PROGRAM main
VAR
	MODBEE_HW_INPUTS0 : MODBEE_HW_INPUTS;
	MODBEE_HW_OUTPUTS0 : MODBEE_HW_OUTPUTS;
	start : bool;
	stop : bool;
	run : bool;
	MODBUS_WRITE0 : MODBUS_WRITE;
	MB_SLAVE_DO01 : bool;
	MB_SLAVE_DO02 : bool;
	MB_SLAVE_DO03 : bool;
	MB_SLAVE_DO04 : bool;
	MB_SLAVE_DO05 : bool;
	MB_SLAVE_DO06 : bool;
	MB_SLAVE_DO07 : bool;
	MB_SLAVE_DO08 : bool;
	MODBUS_READ0 : MODBUS_READ;
	MB_SLAVE_DI01 : bool;
	MB_SLAVE_DI02 : bool;
	MB_SLAVE_DI03 : bool;
	MB_SLAVE_DI05 : bool;
	MB_SLAVE_DI04 : bool;
	MB_SLAVE_DI06 : bool;
	MB_SLAVE_DI07 : bool;
	MB_SLAVE_DI08 : bool;
	MB_WRITE_COILS_DONE : bool;
	MB_READ_COILS_DONE : bool;
	TON0 : TON;
	TON1 : TON;
	TON1_DONE : bool;
	TON0_DONE : bool;
	MODBUS_READ1 : MODBUS_READ;
	MB_READ_REGS_DONE : bool;
	MB_SLAVE_AI01 : int;
	MB_SLAVE_AI02 : int;
	MB_SLAVE_AI03 : int;
	MB_SLAVE_AI04 : int;
	MODBUS_WRITE1 : MODBUS_WRITE;
	MB_WRITE_REGS_DONE : bool;
	MB_SLAVE_AO01 : real;
	MB_SLAVE_AO02 : real;
	MB_SLAVE_AO03 : real;
	MB_SLAVE_AO04 : real;
	MB_SLAVE_AO5 : int;
	MB_SLAVE_AO01_TEMP : int;
	MB_SLAVE_AO02_TEMP : int;
	MB_WRITE_REGS_DONE0 : bool;
END_VAR

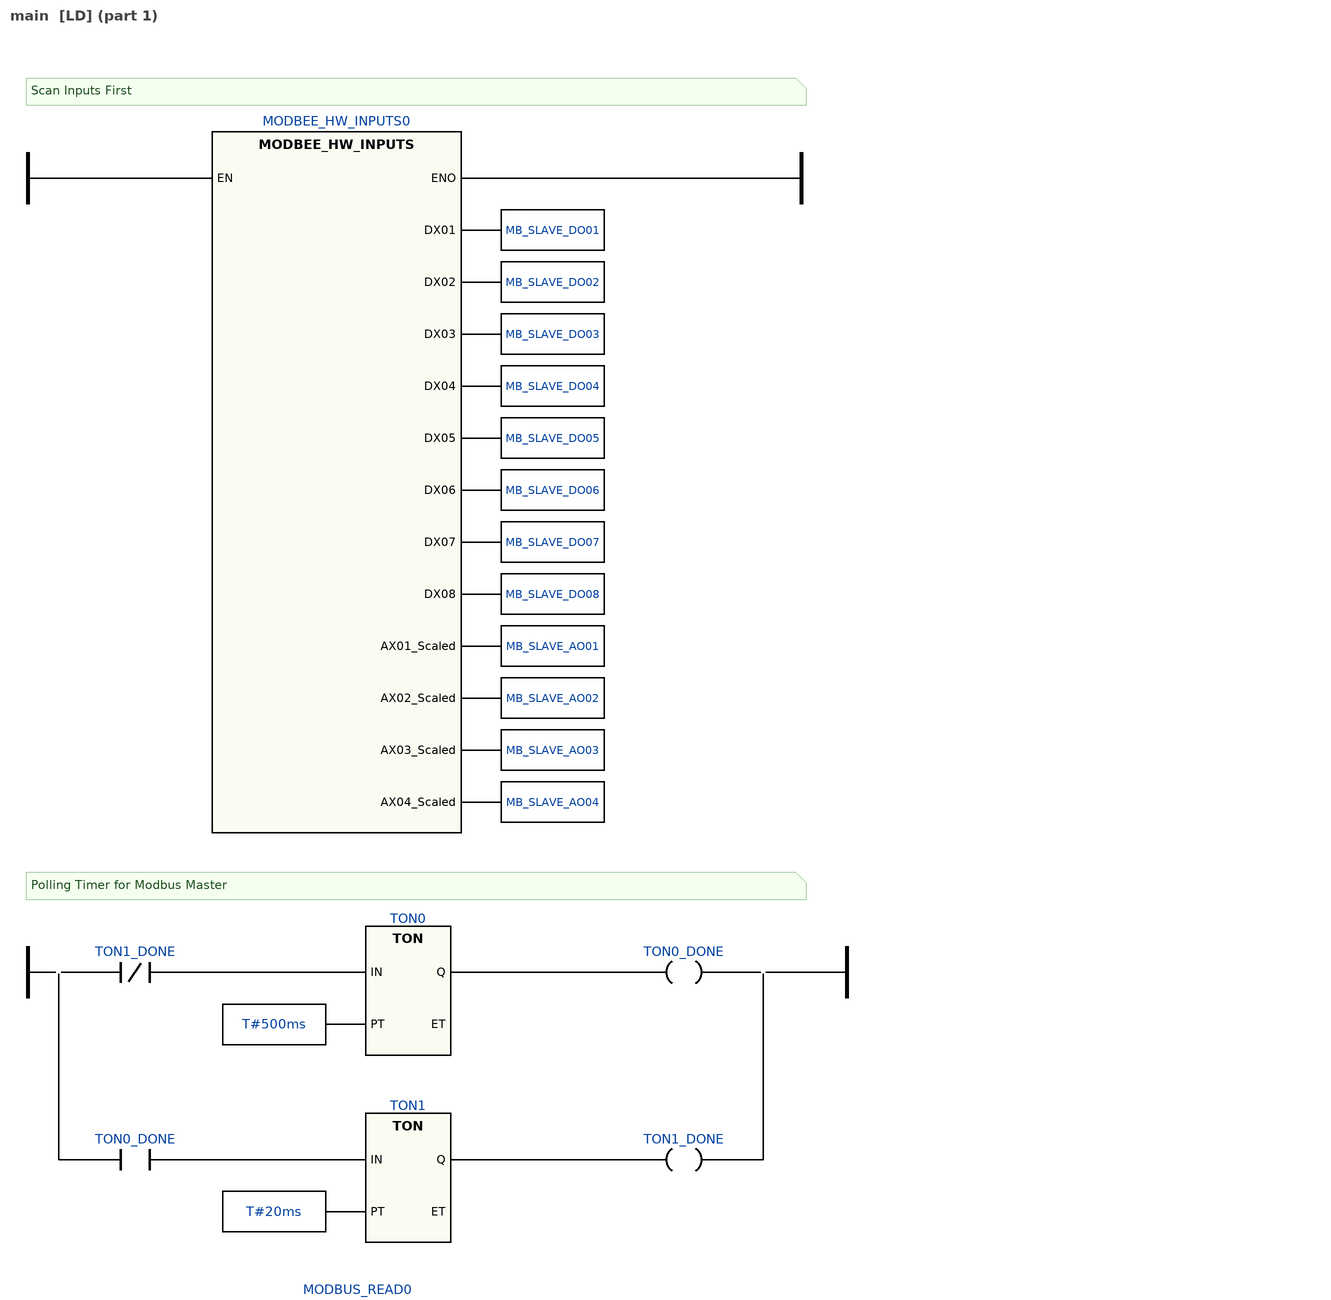
(* LD diagram, written out as Structured Text *)
(* Scan Inputs First *)
MODBEE_HW_INPUTS0();
MB_SLAVE_DO01 := MODBEE_HW_INPUTS0.DX01;
MB_SLAVE_DO02 := MODBEE_HW_INPUTS0.DX02;
MB_SLAVE_DO03 := MODBEE_HW_INPUTS0.DX03;
MB_SLAVE_DO04 := MODBEE_HW_INPUTS0.DX04;
MB_SLAVE_DO05 := MODBEE_HW_INPUTS0.DX05;
MB_SLAVE_DO06 := MODBEE_HW_INPUTS0.DX06;
MB_SLAVE_DO07 := MODBEE_HW_INPUTS0.DX07;
MB_SLAVE_DO08 := MODBEE_HW_INPUTS0.DX08;
MB_SLAVE_AO01 := MODBEE_HW_INPUTS0.AX01_Scaled;
MB_SLAVE_AO02 := MODBEE_HW_INPUTS0.AX02_Scaled;
MB_SLAVE_AO03 := MODBEE_HW_INPUTS0.AX03_Scaled;
MB_SLAVE_AO04 := MODBEE_HW_INPUTS0.AX04_Scaled;
(* Polling Timer for Modbus Master *)
TON0(IN := NOT TON1_DONE, PT := T#500ms);
TON0_DONE := TON0.Q;
TON1(IN := TON0_DONE, PT := T#20ms);
TON1_DONE := TON1.Q;
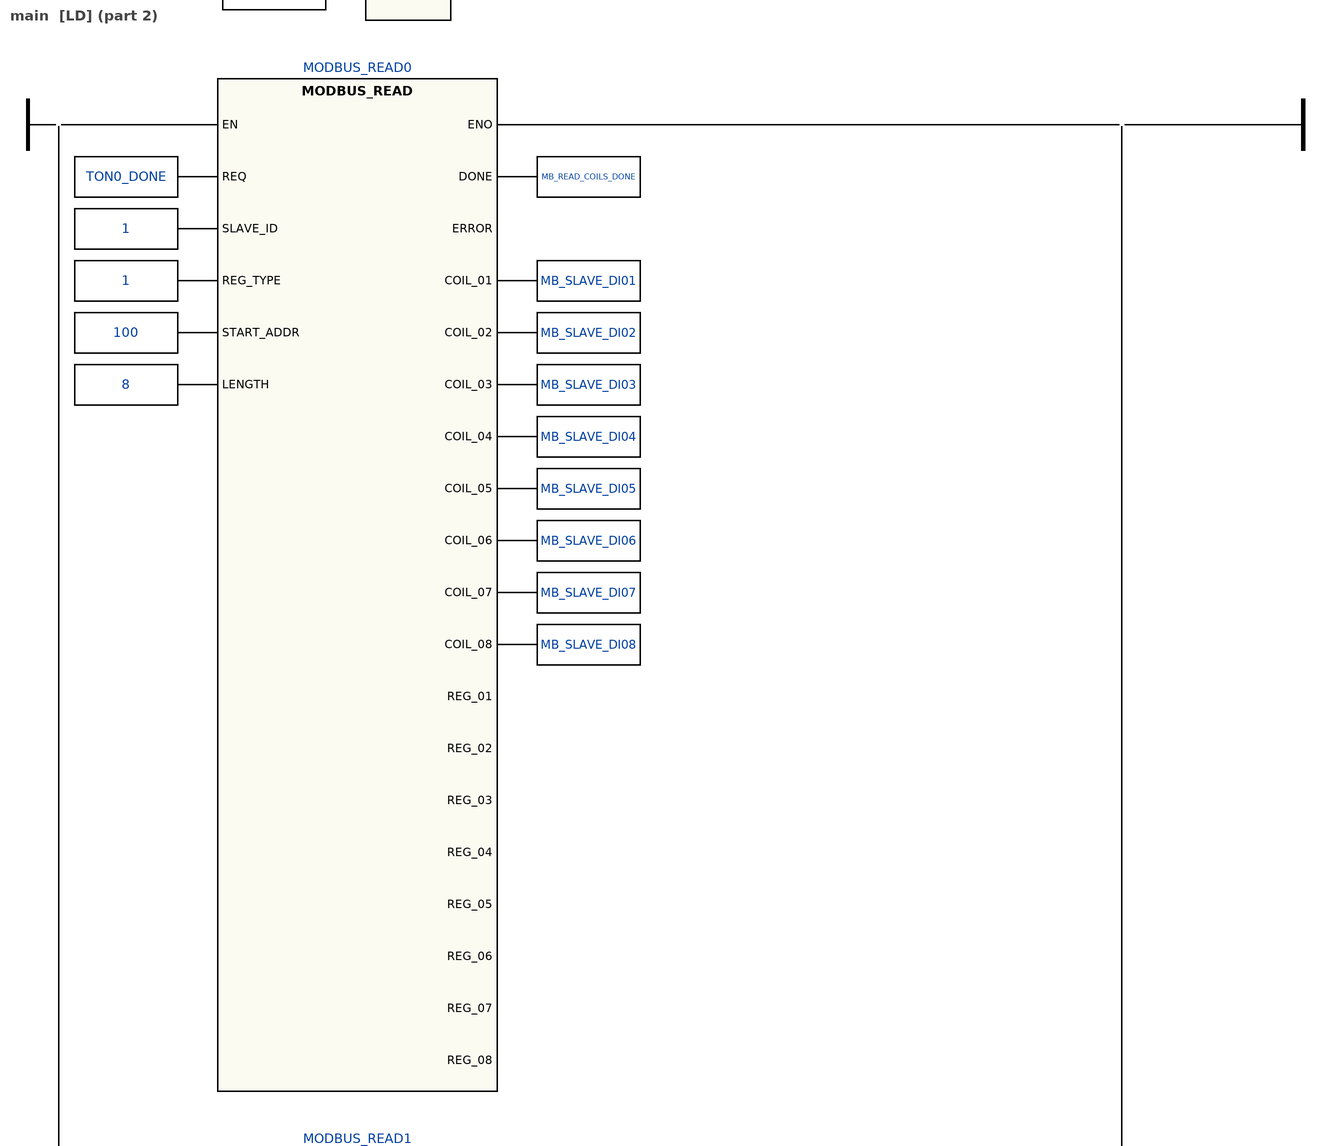
MODBUS_READ0(REQ := TON0_DONE, SLAVE_ID := 1, REG_TYPE := 1, START_ADDR := 100, LENGTH := 8);
MB_READ_COILS_DONE := MODBUS_READ0.DONE;
MB_SLAVE_DI01 := MODBUS_READ0.COIL_01;
MB_SLAVE_DI02 := MODBUS_READ0.COIL_02;
MB_SLAVE_DI03 := MODBUS_READ0.COIL_03;
MB_SLAVE_DI04 := MODBUS_READ0.COIL_04;
MB_SLAVE_DI05 := MODBUS_READ0.COIL_05;
MB_SLAVE_DI06 := MODBUS_READ0.COIL_06;
MB_SLAVE_DI07 := MODBUS_READ0.COIL_07;
MB_SLAVE_DI08 := MODBUS_READ0.COIL_08;
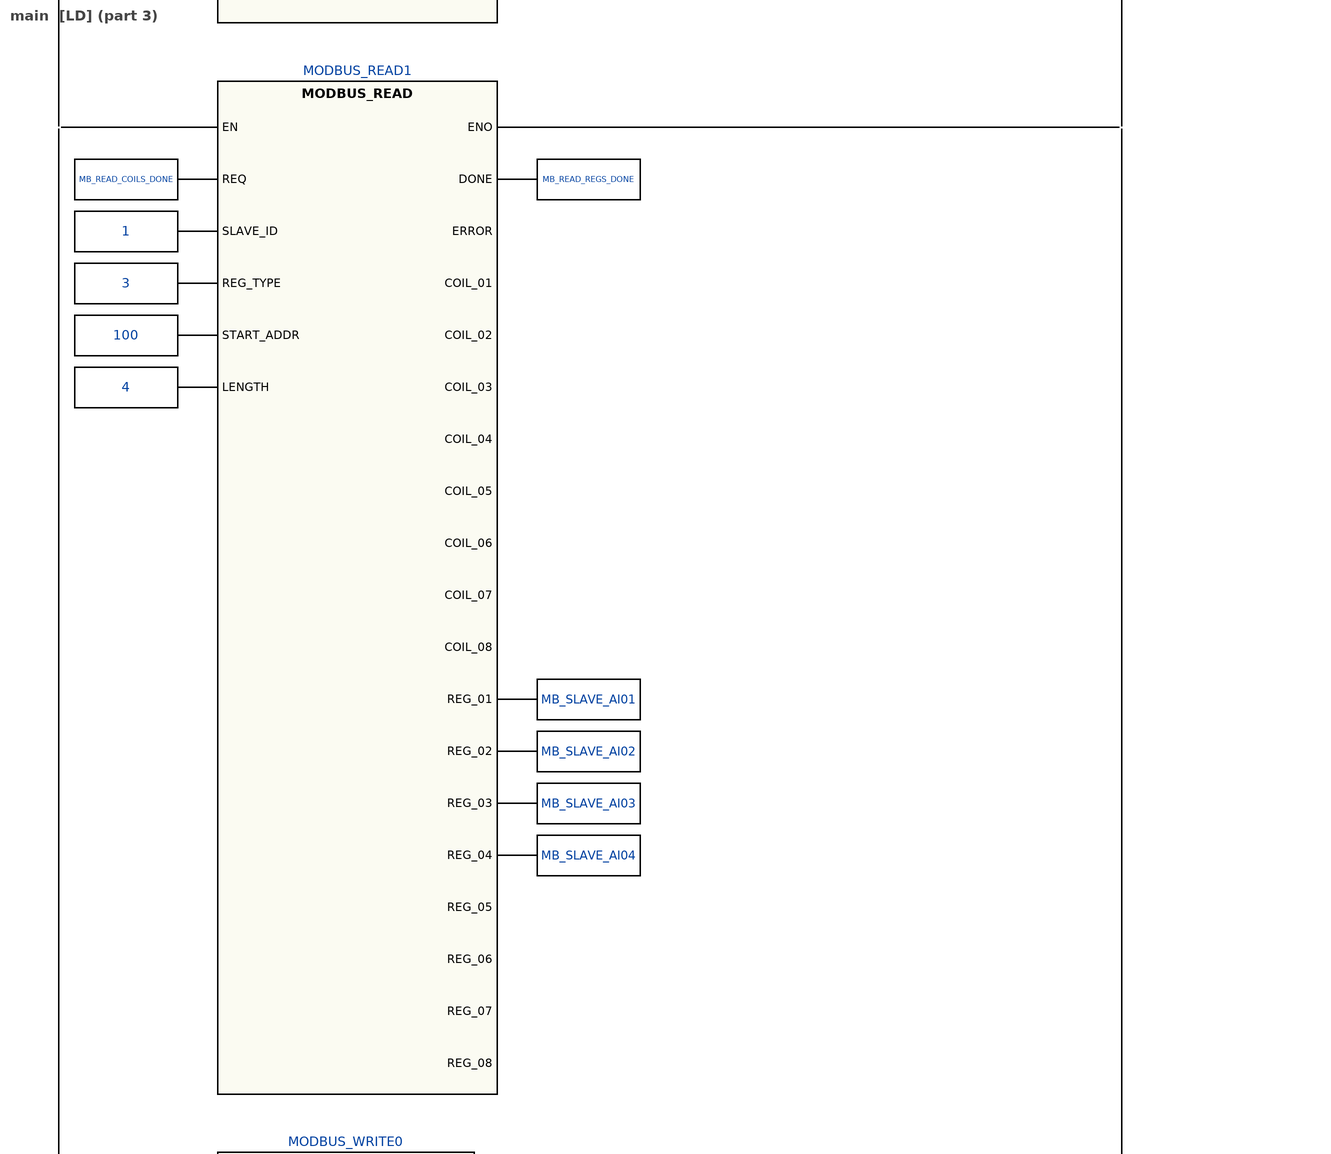
MODBUS_READ1(REQ := MB_READ_COILS_DONE, SLAVE_ID := 1, REG_TYPE := 3, START_ADDR := 100, LENGTH := 4);
MB_READ_REGS_DONE := MODBUS_READ1.DONE;
MB_SLAVE_AI01 := MODBUS_READ1.REG_01;
MB_SLAVE_AI02 := MODBUS_READ1.REG_02;
MB_SLAVE_AI03 := MODBUS_READ1.REG_03;
MB_SLAVE_AI04 := MODBUS_READ1.REG_04;
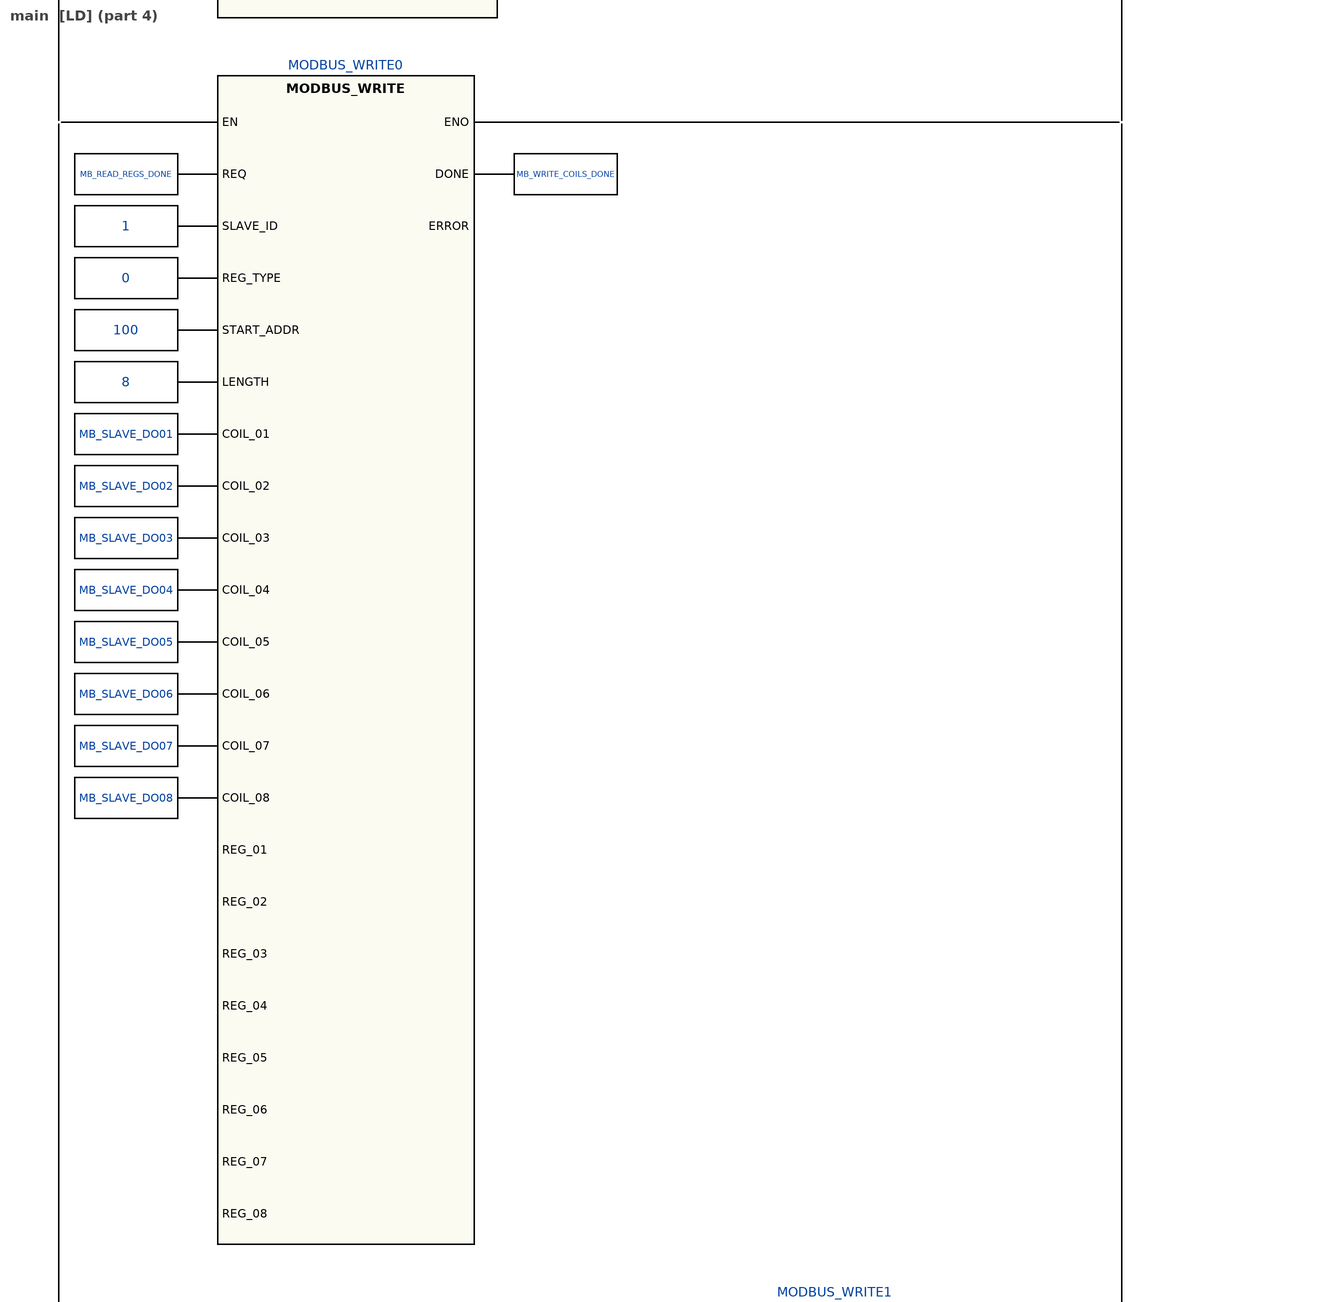
MODBUS_WRITE0(REQ := MB_READ_REGS_DONE, SLAVE_ID := 1, REG_TYPE := 0, START_ADDR := 100, LENGTH := 8, COIL_01 := MB_SLAVE_DO01, COIL_02 := MB_SLAVE_DO02, COIL_03 := MB_SLAVE_DO03, COIL_04 := MB_SLAVE_DO04, COIL_05 := MB_SLAVE_DO05, COIL_06 := MB_SLAVE_DO06, COIL_07 := MB_SLAVE_DO07, COIL_08 := MB_SLAVE_DO08);
MB_WRITE_COILS_DONE := MODBUS_WRITE0.DONE;
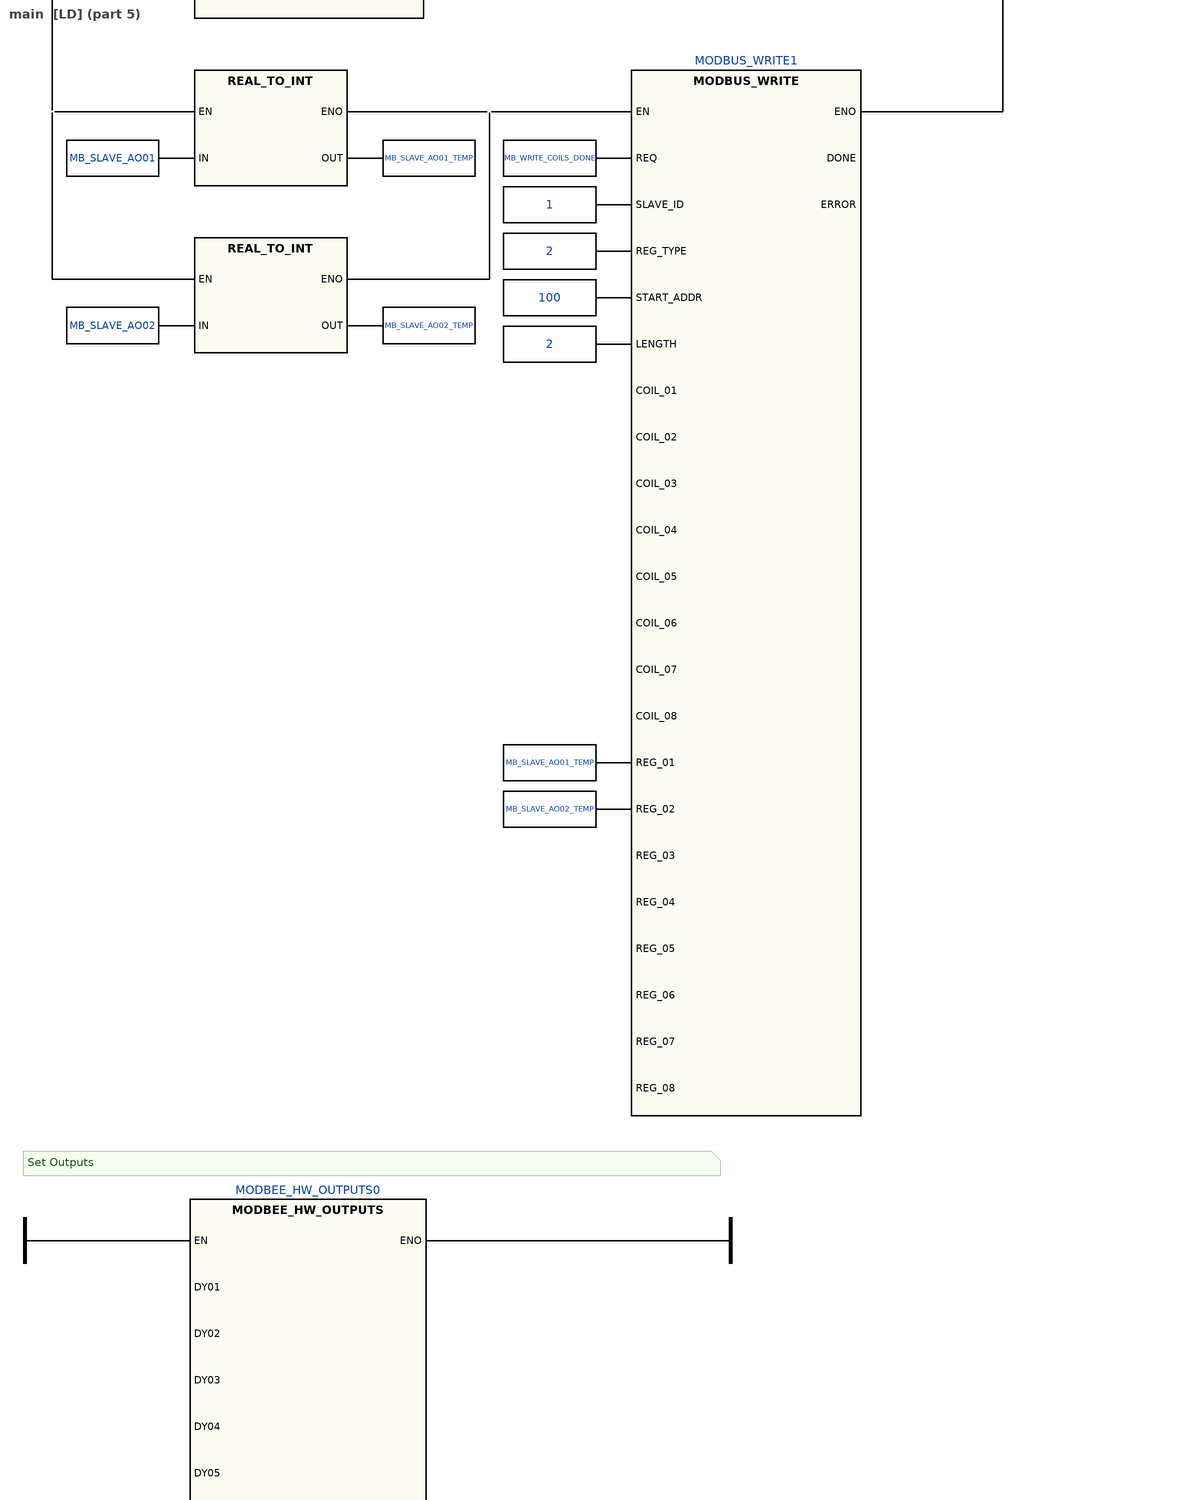
MB_SLAVE_AO01_TEMP := REAL_TO_INT(MB_SLAVE_AO01);
MB_SLAVE_AO02_TEMP := REAL_TO_INT(MB_SLAVE_AO02);
MODBUS_WRITE1(REQ := MB_WRITE_COILS_DONE, SLAVE_ID := 1, REG_TYPE := 2, START_ADDR := 100, LENGTH := 2, REG_01 := MB_SLAVE_AO01_TEMP, REG_02 := MB_SLAVE_AO02_TEMP);
(* Set Outputs *)
MODBEE_HW_OUTPUTS0();
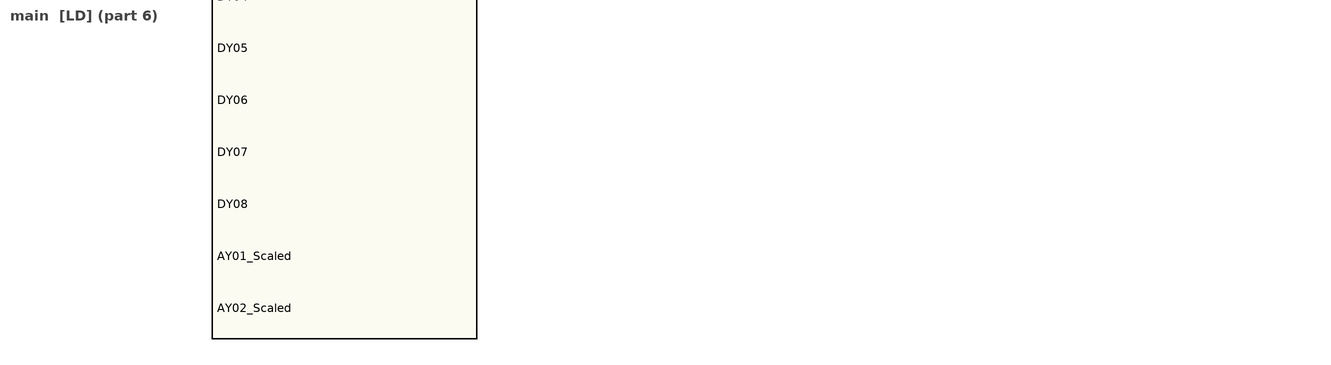
END_PROGRAM
